// TIA Portal V17 export
// export: Created 2023-06-16T13:19:14.8358831Z, ExportSetting WithDefaults, DisplayName Totally Integrated Automation Portal, DisplayVersion V17, DisplayName TIA Portal Openness, DisplayVersion V17, DisplayName TIA Portal Version Control Interface, DisplayVersion V17, DisplayName STEP 7 Professional, DisplayVersion V17, DisplayName STEP 7 Safety, DisplayVersion V17, DisplayName WinCC Advanced, DisplayVersion V17
VAR_GLOBAL   // PLC tag table "IOVartab"
   "Input test" AT %I0.0 : Bool;
   "Output test" AT %Q0.0 : Bool;
END_VAR
